// TIA Portal V18 export
TYPE "LGasp_type_Bck_comandi"
// stored: IsFailsafeCompliant false
   STRUCT
      cmdbool00 : Array[1..32] of Bool;
      cmdbool01 : Array[1..32] of Bool;
      cmdbool02 : Array[1..32] of Bool;
      cmdbool3 : Array[1..32] of Bool;
      cmdint : Array[1..32] of Int;
      cmddint : Array[1..32] of DInt;
      cmdlreal : Array[1..32] of LReal;
      cmdstring : Array[1..32] of WString;
   END_STRUCT;
   // // cmdbool00[1] : richiesta trasferimento lista produzione
   // // cmdbool00[2] : ok ad aggiornamento trasferimento valori DS
   // // cmdbool00[3] : spare
   // // cmdbool00[4] : richiesta svuotamento
   // // cmdbool00[5] : abilitazione trasferimento righe di produzione
   // // cmdbool00[6] : spare
   // // cmdbool00[7] : compila lista (PC SET / RESET)
   // // cmdbool00[8] : elimina elemento lista tagli (PC SET, PLC RESET)
   // // cmdbool00[9] : Pulsante cancelli pezzi fatti (PC SET, PLC RESET) (previsione)
   // // cmdbool00[10] : Segnale lista online modificata (PC SET, PC RESET al download successivo)
   // // cmdbool00[11] : Pulsante reset completo lista produzione (PC SET, PLC RESET)
   // // cmdbool00[12] : Segnale life bit da PC (PC SET - PLC RESET)
   // // cmdbool00[13] : Cancellazione completa lista tagli
   // // cmdbool00[14] : Ripristina lista profila
   // // cmdbool00[15] : Conferma visualizzazione finestra inserimento lamiera
   // // cmdbool00[17] : Conferma salvataggio correttori profila
   // // cmdbool00[18] : Invio dati Approntamento profila eseguito
   // // cmdbool00[19] : Risposta approntamento completato
   // // cmdbool00[20] : Comando sincronizzazione profila
   // // cmdbool00[21] : Comando invio correttori approntamento assi inviato
   // // cmdbool00[22] : Comando Svuotamento scarico
   // // cmdbool00[23] : Abilitazione nervaturaAbilitazione film su lamiera
   // // cmdbool00[24] : Abilitazione nervaturaAbilitazione film su lamiera
   // // cmdbool00[32] : abilita pulsante svuotamento da PLC
   // // cmdbool01[1] : Prodotto Impilabile (0: No, 1: Si)
   // // cmdbool01[2] : Prodotto NON forato (0: No, 1: Si)
   // // cmdbool01[3] : Prodotto Rastremato (0: No, 1: Si)
   // // cmdbool01[10] : Conferma posizionamento stampo mobile P04 (210100012)
   // // cmdint[1] : Numero di righe pagina di produzione dainviare
   // // cmdint[2] : Tipo profilo in approntamento (da codificare)
   // // cmdint[3] : Impilabile (0: No, 1: Si)
   // // cmdint[4] : Tipo lavorazione specifica del prodotto (Spare05) a partire da 210100068
   // // cmdint[7] : 1=cumulativo warning vita punzoni, 2=cumulativo allarme vita punzone, reset da PC
   // // cmdlreal[1] : Spessore
   // // cmdlreal[2] : Override 1- 100 %
   // // cmdlreal[3] : Correttore lunghezze
   // // cmdlreal[4] : Sviluppo reale Coil per centraggio
   // // cmdlreal[5] : Base nominale profilo selezionato
   // // cmdlreal[6] : Altezza nominale profilo selezionato
   // // cmdlreal[7] : Sfrido taglio
   // // cmdlreal[8] : Peso specifico materiale (g/cm3)
   // // cmdlreal[9] : Correttore offset taglio
   // // cmdlreal[10] : Dimensione aletta
   // // cmdlreal[11] : Correttore ruota metrica taglio
   // // cmdstring[1] : visualizzazione produzione in lavoro
   // // cmdstring[2] : visualizzazione prossima produzione
   // // cmdstring[3] : Codice colata
END_TYPE
